TYPE ST_HomeAbsSwitch :
STRUCT
	pSignalInput		: POINTER TO BOOL;	
	SensorEdgeSignal 	: eHomeModeOption;	
	Trigger_Direction	: eHomeModeOption;
END_STRUCT
END_TYPE

(* stored: Version 1.1.0.1, ProductVersion 3.1.4024.3
   DUT ST_HomeAbsSwitch: Id {e50872af-4c6c-0dd3-215d-cc762ccccace} *)
